KUKA KRL program: chk_w3_grp2_clo.src

&ACCESS RVO1
&COMMENT Check GRP ACTROS Z2 CLOSE
DEF chk_w3_grp2_clo( )

;//---- Start User-------
;Aguardando posicao de gripper fechado

$TIMER[10] = 0
$TIMER_STOP[10] = FALSE

WAIT FOR (NOT $IN[11] AND NOT $IN[13])
WAIT FOR ($IN[12] AND $IN[14])

$TIMER_STOP[10] = TRUE
$TIMER[10] = 0

;//---- End User-------

END
